RoboDK station: Polar_MH6.rdk

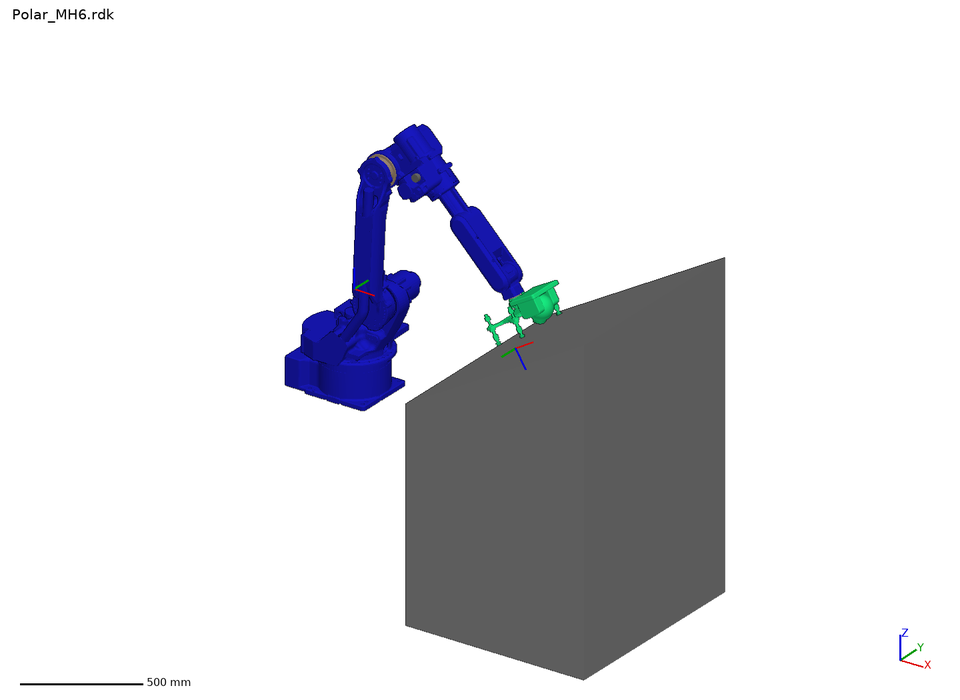
[picture v0: the station drawn from its stored meshes, robots at their saved joint values, targets as dots, program paths as lines]
Station L2 (saved by RoboDK 5.9.3). Poses are relative to the parent item; angles as X-Y-Z fixed-axis rotations.
  - frame Motoman MH6 Base at (0, 0, 450) mm
    - robot Motoman MH6: 6 axes, payload 6 kg, reach 1422 mm, repeatability 0.08 mm, weight 130 kg
        modified DH rows (alpha deg, a mm, theta deg, d mm): 0, 0, 0, 450; -90, 152, -90, 0; 0, 614, 0, 0; -90, 155, 0, 640; 90, 0, 90, 0; -90, 0, 0, 95
        base shift (0, 0, -450) mm
        joint limits [-170, -90, -175, -180, -45, -360] to [170, 155, 250, 180, 225, 360]; home [0, 0, 0, 0, 0, 0]; saved at [1.171, 2.819, -43.46, 2.465, 76.262, -3.408]
      - tool Ventosas, TCP at (0, 0, 190) mm, size 250 x 290 x 148 mm
    - frame Frame_from_Target1 at (823.2, -34.49, -21.13) mm, rotated rx -180 ry -30 rz 0 deg
  - object CAJA2 at (1600, 500, 300) mm, rotated rx 180 ry 0 rz 0 deg, size 886.4 x 1000 x 1511.7 mm, geometry from CAJA2.stp
  - Python program Polar_Names (listed below)

--- Python program Polar_Names ---
from robodk.robolink import *    # API para comunicarte con RoboDK
from robodk.robomath import *    # Funciones matemáticas
import math
from matplotlib.textpath import TextPath
from matplotlib.font_manager import FontProperties
import numpy as np

# ------------------------------------------------
# Inicialización RoboDK
# ------------------------------------------------
RDK = Robolink()
robot = RDK.ItemUserPick("Selecciona un robot", ITEM_TYPE_ROBOT)
#if not robot.Valid():
#    raise Exception("No se ha seleccionado un robot válido.")

# Conectar al robot físico
#if not robot.Connect():
#    raise Exception("No se pudo conectar al robot. Verifica que esté en modo remoto y que la configuración sea correcta.")

# Confirmar conexión
#if not robot.ConnectedState():
#    raise Exception("El robot no está conectado correctamente. Revisa la conexión.")

#print("Robot conectado correctamente.")

frame_name = "Frame_from_Target1"
frame = RDK.Item(frame_name, ITEM_TYPE_FRAME)
# Asignamos este frame al robot
robot.setPoseFrame(frame)
# Usamos la herramienta activa
robot.setPoseTool(robot.PoseTool())

robot.setSpeed(500)
robot.setRounding(5)

z_surface = 0
z_safe = -50
home = transl(0, 0, z_surface + z_safe)
home_abs = transl(0, 0, z_surface - 300)

# ------------------------------------------------
# draw_text_with_path: reflejo + rotación (plano)
# ------------------------------------------------
def draw_text_with_path(text, x_offset, y_offset, z,
                        font_size=75, font_name='Arial',
                        rotation_deg=90, mirror_x=True):
    """
    Dibuja texto usando TextPath aplicando:
      - copia writable de vértices,
      - reflejo en X (mirror_x),
      - rotación en el plano XY de 'rotation_deg' grados.
    rotation_deg: ángulo en grados (ej. 90 para girarlo 90°).
    """
    fp = FontProperties(family=font_name, size=font_size)
    tp = TextPath((0, 0), text, prop=fp)

    # copiar para evitar read-only
    vertices = tp.vertices.copy()
    codes = tp.codes.copy() if tp.codes is not None else None

    # 1) reflejo en X si se requiere (arregla "texto en espejo")
    if mirror_x:
        vertices[:, 0] = -vertices[:, 0]

    # 2) rotación en el plano XY
    theta = math.radians(rotation_deg)
    rot = np.array([[math.cos(theta), -math.sin(theta)],
                    [math.sin(theta),  math.cos(theta)]])
    vertices = vertices @ rot.T  # aplicar rotación

    # seguridad: si no hay vértices, salir
    if vertices.shape[0] == 0:
        return

    # mover a punto inicial en modo seguro (arriba)
    start_x = x_offset + float(vertices[0, 0])
    start_y = y_offset + float(vertices[0, 1])
    robot.MoveL(transl(start_x, start_y, z_surface + z_safe))

    # bajar a superficie
    robot.MoveL(transl(start_x, start_y, z))

    # recorrer vértices
    n = len(vertices)
    for i in range(1, n):
        vx = x_offset + float(vertices[i, 0])
        vy = y_offset + float(vertices[i, 1])

        if codes is not None and codes[i] == 1:  # MOVETO -> levantar y desplazar
            prev_x = x_offset + float(vertices[i - 1, 0])
            prev_y = y_offset + float(vertices[i - 1, 1])
            robot.MoveL(transl(prev_x, prev_y, z_surface + z_safe))
            robot.MoveL(transl(vx, vy, z_surface + z_safe))
            robot.MoveL(transl(vx, vy, z))
        else:
            robot.MoveL(transl(vx, vy, z))

    # subir al terminar
    last_x = x_offset + float(vertices[-1, 0])
    last_y = y_offset + float(vertices[-1, 1])
    robot.MoveL(transl(last_x, last_y, z_surface + z_safe))


# ------------------------------------------------
# Curva polar (sin cambios)
# ------------------------------------------------
def polar(x_offset, y_offset, A, n):
    num_points = 180
    full_turn = 2 * math.pi
    for i in range(num_points + 1):
        t = i / num_points
        theta = full_turn * t
        r = A * (4 + math.cos(n * theta) + math.sin(n * theta) ** 2)
        x = r * math.cos(theta) + x_offset
        y = r * math.sin(theta) + y_offset
        robot.MoveL(transl(x, y, z_surface))
    robot.MoveL(transl(x, y, z_surface + z_safe))


# ------------------------------------------------
# Programa principal (ejemplo)
# ------------------------------------------------
def main():
    robot.MoveJ(home_abs)
    robot.MoveJ(home)

    # dibujar rosa polar
    polar(230, 0, 30, 5)

    # Opciones: rotation_deg=90 gira 90° para ver horizontal cuando se escribía en "cara"
    # mirror_x=True corrige efecto espejo si aparece
    draw_text_with_path("Santiago", 150 - 120, -120, z_surface,
                        font_size=75, rotation_deg=-90, mirror_x=True)

    # bajar "Samuel" más
    draw_text_with_path("Samuel", 100 - 180, -120, z_surface,
                        font_size=75, rotation_deg=-90, mirror_x=True)

    robot.MoveJ(home)
    robot.MoveJ(home_abs)
    print("¡Terminado!")

if __name__ == "__main__":
    main()
